FUNCTION_BLOCK PistonForce
VAR_INPUT
	PistonVelocity : LREAL;
	Piston_Position : LREAL;
	PressureBoreSide : LREAL;
	PressureRodSide : LREAL;
	Aa : LREAL;
	Ab : LREAL;
	param : HydraulicCylinder;
END_VAR
VAR_OUTPUT
	F_Piston : LREAL;
END_VAR
VAR
	y_tmp : LREAL;
END_VAR

//Hydraulic Force [N]
F_Hydraulic := param.PressureBoreSide * param.Aa - param.PressureRodSide * param.Ab;


//Upper Stroke Limit Contact Force [N]




//Lower Stroke Limit Contact Force [N]




//Stribeck Friction Force [N]
y_tmp := EXP((PistonVelocity * 250.0) * 2.0);
y_tmp := (y_tmp - 1.0) / (y_tmp + 1.0);
Stribeck_F := (((EXP(( -(PistonVelocity * y_tmp)) / 0.02) * 500.0) + 75.0) * y_tmp) + (PistonVelocity * 1500.0);




//Piston Force Total [N]
F_Piston := F_Hydraulic - F_Upper_Stroke_Limit + F_Lower_Stroke_Limit - F_Stribeck_Friction;




//IF higher/lower than value formula for PLC:
//IF PistonPosition >= param.xMax THEN 
//	PistonPosition := param.xMax;
//ELSIF PistonPosition <= 0 THEN 
//	PistonPosition := 0;
//END_IF;

END_FUNCTION_BLOCK

(* stored: Version 1.1.0.1, ProductVersion 3.1.4024.9
   POU PistonForce: Id {2815a2de-522e-4f8d-ac11-c59cbc1ac2b7}, SpecialFunc None *)
